FUNCTION_BLOCK FB_ButtonEnable
VAR_INPUT
	SET:	BOOL;
	RESET:	BOOL;
END_VAR
VAR_OUTPUT
	Q: BOOL;
END_VAR
VAR
	trigger:	R_TRIG;
	ftrigger:	F_TRIG;
	state:		RS;
END_VAR

trigger(CLK := SET);
ftrigger(CLK := SET);
state(SET := trigger.Q AND NOT Q,
	RESET1 := RESET OR (trigger.Q AND Q),
	Q1 => Q);

END_FUNCTION_BLOCK

(* stored: Version 1.1.0.1, ProductVersion 3.1.4024.6
   POU FB_ButtonEnable: Id {3211ceeb-9597-41c3-8547-3ce80543891d}, SpecialFunc None *)
